FUNCTION_BLOCK SFC1 (* Basic Function Block Type *)
  (* Standard: 61499-2 *)
  (* Version 0.2, 2003-12-04, JHC, Rockwell Automation, Renamed for better indexing. *)
  (* Version 0.1, 2002-11-05, JHC, Rockwell Automation, Corrected missing ST element in Algorithm REQ. *)
  (* Version 0.0, 2000-05-30, JHC, Rockwell Automation *)
  (* Compiler header: package fb.rt.pnp; *)
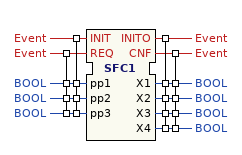
  EVENT_INPUT
    INIT WITH pp1, pp2, pp3; (* Initialization Request *)
    REQ WITH pp1, pp2, pp3; (* Normal Execution Request *)
  END_EVENT
  EVENT_OUTPUT
    INITO WITH X1, X3, X2, X4; (* Initialization Confirm *)
    CNF WITH X1, X2, X3, X4; (* Execution Confirmation *)
  END_EVENT
  VAR_INPUT
    pp1 : BOOL; (* Input event qualifier *)
    pp2 : BOOL;
    pp3 : BOOL;
  END_VAR
  VAR_OUTPUT
    X1 : BOOL; (* Output event qualifier *)
    X2 : BOOL;
    X3 : BOOL;
    X4 : BOOL;
  END_VAR
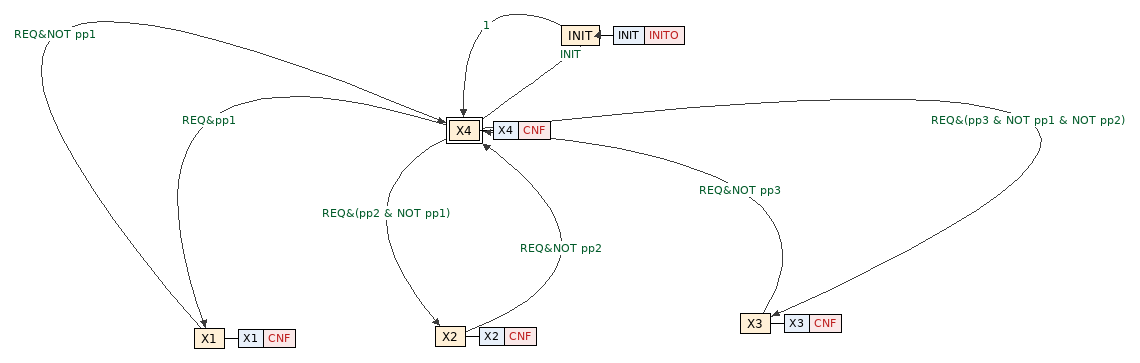
  EC_STATES
    X4 : X4 -> CNF; (* Initial State *)
    INIT : INIT -> INITO; (* Initialization *)
    X1 : X1 -> CNF; (* Normal execution *)
    X2 : X2 -> CNF;
    X3 : X3 -> CNF;
  END_STATES
  EC_TRANSITIONS
    X4 TO INIT := INIT;
    INIT TO X4 := 1;
    X4 TO X1 := REQ&pp1;
    X4 TO X2 := REQ&(pp2 & NOT pp1);
    X4 TO X3 := REQ&(pp3 & NOT pp1 & NOT pp2);
    X1 TO X4 := REQ&NOT pp1;
    X2 TO X4 := REQ&NOT pp2;
    X3 TO X4 := REQ&NOT pp3;
  END_TRANSITIONS
  ALGORITHM INIT IN ST: (* Initialization algorithm *)
X1:=false;
X2:=false;
X3:=false;
X4:=false;
System.out.println("SFC1: INIT");
  END_ALGORITHM
  ALGORITHM REQ IN ST: (* Normally executed algorithm *)

  END_ALGORITHM
  ALGORITHM X4 IN ST:
X4:=true;
IF NOT pp1 THEN
X1:=false;
END_IF
IF NOT pp2 THEN
X2:=false;
END_IF
IF NOT pp3 THEN
X3:=false;
END_IF
System.out.println("SFC1: X4");
  END_ALGORITHM
  ALGORITHM X1 IN ST:
X1:= true;
X4:=false;
System.out.println("SFC1: X1");
  END_ALGORITHM
  ALGORITHM X2 IN ST:
X2:= true;
X4:=false;
System.out.println("SFC1: X2");
  END_ALGORITHM
  ALGORITHM X3 IN ST:
X3:= true;
X4:=false;
System.out.println("SFC1: X3");
  END_ALGORITHM
END_FUNCTION_BLOCK
